FUNCTION_BLOCK FB_Blink
VAR_INPUT
	msTime		:UDINT;	
END_VAR
VAR_OUTPUT
	sig		:BOOL;
END_VAR
VAR
	timeCounter		:UDINT;
	rtc				:GETCPUACCOUNT;
END_VAR

	
//
	rtc(cpuAccountDW=> );

	IF rtc.cpuAccountDW - timeCounter >= msTime*10000 THEN 
		sig := NOT sig;
		timeCounter := rtc.cpuAccountDW;
	END_IF

END_FUNCTION_BLOCK

(* stored: Version 1.1.0.1, ProductVersion 3.1.4022.16
   POU FB_Blink: Id {eb17dbb5-fa83-4aea-94bb-b4b31df5a416}, SpecialFunc None *)
